{attribute 'qualified_only'}
VAR_GLOBAL
	
	safetyOK : BOOL;
	i_KUKAStatus : INT;
END_VAR

(* stored: Version 1.1.0.1, ProductVersion 3.1.4024.12
   GVL GVL: Id {f69daea1-3c7b-453a-b10c-118c41e8a30e} *)
